FUNCTION_BLOCK FB_RtdSensor EXTENDS FB_ComponentBase IMPLEMENTS I_TempSensor
VAR
	_InSimulation : BOOL;
END_VAR

//{warning 'Add method implementation '}
METHOD CyclicLogic
IF _InSimulation THEN
	CyclicSimulate();
ELSE
	;
END_IF
END_METHOD

METHOD CyclicSimulate
VAR_INPUT
END_VAR
END_METHOD

PROPERTY InSimulation : BOOL
GET
InSimulation := _InSimulation;
END_GET
SET
_InSimulation := InSimulation;
END_SET
END_PROPERTY

{warning 'Add method implementation '}
METHOD Reset : BOOL
END_METHOD

{warning 'Add property implementation'}
PROPERTY Temp : LREAL
GET
END_GET
END_PROPERTY

END_FUNCTION_BLOCK

(* stored: Version 1.1.0.1
   POU FB_RtdSensor: Id {2e353b4b-b106-4727-b887-bf1f9517787d}, SpecialFunc None
   Method CyclicLogic: Id {5c28ce19-f03b-4481-9569-2cafac0a0828}
   Method CyclicSimulate: Id {7e91be32-ae97-48c8-9110-6773dfddac1e}
   Property InSimulation: Id {0e42623d-33ad-439a-a09f-3e627d2ee02d}
   Get Get: Id {384af5e3-4117-41c7-840a-8b82036b671b}
   Set Set: Id {537e02dd-67b1-4c08-9868-c907bb468574}
   Method Reset: Id {66ed542f-4215-4de9-a84c-fbc1d2ef08b8}
   Property Temp: Id {15551044-a344-41f3-86cc-c8cdf380c97d}
   Get Get: Id {4f7d9504-81a8-4ef7-9285-a686f0e15403} *)
